PROGRAM MAIN
VAR
    bLed : BOOL;
    fbTimer : TON;
END_VAR

fbTimer(IN := NOT fbTimer.Q, PT := T#1S);

IF fbTimer.Q THEN
    bLed := NOT bLed;
END_IF

END_PROGRAM

(* stored: Version 1.1.0.1
   POU MAIN: Id {2a67b1bd-69a0-4a73-bbd9-c4d61c319d4e}, SpecialFunc None *)
